// TIA Portal V20 export
TYPE "zp_CITI_Features"
// stored: Access Published, Namespace CITI_Logic
   STRUCT
      Map_Enable : Bool;
      RemoteConfig_En : Bool := FALSE;
      SL_Enable : Bool := FALSE;
      AndonMap_En : Bool := FALSE;
      Fault_Data : Bool := FALSE;
      StringData : Bool := FALSE;
      Blocked : Bool := FALSE;
      Starved : Bool := FALSE;
      Loading : Bool := FALSE;
      Unloading : Bool := FALSE;
      Idle : Bool := FALSE;
      Wait_1 : Bool := FALSE;
      Wait_2 : Bool := FALSE;
      Wait_3 : Bool := FALSE;
      Wait_4 : Bool := FALSE;
      OperatorOvercycle1 : Bool := FALSE;
      OperatorOvercycle2 : Bool := FALSE;
      ManualMode : Bool := FALSE;
      QualityCheck : Bool := FALSE;
      ToolChange : Bool := FALSE;
      MaterialLow : Bool := FALSE;
      EnergyConservation : Bool := FALSE;
      SafetyChecksum : Bool := FALSE;
      Bypass : Bool := FALSE;
      Bypass_Cnt : Bool := FALSE;
      GoodPart_Cnt : Bool := FALSE;
      RejectPart_Cnt : Bool := FALSE;
      PUN : Bool := FALSE;
      BufferBypass : Bool := FALSE;
      PartType : Bool := FALSE;
      FTQ : Bool := FALSE;
      AndonHold : Bool := FALSE;
      Cycle : Bool := FALSE;
      OnlinePallet_Cnt : Bool := FALSE;
      OnlineEmptyPallet_Cnt : Bool := FALSE;
      OfflinePallet_Cnt : Bool := FALSE;
      Buffer_Cnt : Bool := FALSE;
      PalletID : Bool := FALSE;
      ProcessRetry_Cnt : Bool := FALSE;
      SPC_Cnt : Bool := FALSE;
      GM_PN : Bool := FALSE;
      Opt_Data : Bool := FALSE;
      CMM_Data : Bool := FALSE;
      "Filter Data" : Bool := FALSE;
      Tank_Level : Bool := FALSE;
      Pump_Back_Level : Bool := FALSE;
      Tank_Coolant_Temp : Bool := FALSE;
      DryCycle_Mode : Bool := FALSE;
      Using_GCCS_Template : Bool := FALSE;
   END_STRUCT;
END_TYPE
